	IF pVeData <> 0 THEN
		iDatatypeSize := SIZEOF(ptr^);
		iDatatypeSize := 24;
        ptr := ADR(pVeData^)  +  24  * nVEIndex + (iDatatypeSize * (nArrayIndex));
        ptr^ := val; (* successfully completed return *)
		HLI3_SetVEChannelStringValue := TRUE;
	END_IF
END_IF

END_FUNCTION

// CNC/6 BlockSearch/HLI3_BlockSearch
FUNCTION_BLOCK HLI3_BlockSearch
VAR_INPUT
	/// Number of channel 
	nChanIdx: INT;
	/// interface values 
	BlockSearch: ST_BlockSearch;
END_VAR
VAR_IN_OUT
	/// Edge signal 
	bStartWrite: BOOL;
	/// Edge signal 
	bStartRead: BOOL;
END_VAR
VAR_OUTPUT
	Busy: BOOL;
	Err: BOOL;
	nErrorState: UINT;
	/// interface values 
	nActType: INT;
	fActDistance: LREAL;
	bActAutoReturn: BOOL;
	nActDeviationMax: UDINT;
	nActBlockNumber: DINT;
	nActPass: DINT;
	nActBlockCount: DINT;
	/// current values 
	actualBlockNumber: DINT := 0;
	actualBlockCount: UDINT := 0;
	actualBlockCount_AfterReset: UDINT := 0;
	coveredDistance: DINT;
	coveredDistance_AfterReset: DINT := 0;
END_VAR
VAR
	bReadStarted: BOOL;
	bWriteStarted: BOOL;
	rtStartRead: R_TRIG;
	rtStartWrite: R_TRIG;
	writeType: WriteBsType;
	readType: ReadBsType;
	writeDistance: WriteBsCoveredDistance;
	readDistance: ReadBsCoveredDistance;
	writeAutoReturn: WriteBsAutoReturn;
	readAutoReturn: ReadBsAutoReturn;
	writeDeviationMax: WriteBsDeviationMax;
	readDeviationMax: ReadBsDeviationMax;
	writeBlockNumber: WriteBsBlockNumber;
	ReadBlockNumber: ReadBsBlockNumber;
	writeBlockCount: WriteBsBlockCount;
	ReadBlockCount: ReadBsBlockCount;	
	writePass: WriteBsPass;
	readPass: ReadBsPass;
	nChannelIdxGrp: UDINT;
	/// Timer to read axisposition cyclically        
	Timer: TON;
	actualcoveredDistance: BOOL;
	ChannelMode: UDINT;
	BlockSearchStart: BOOL;
END_VAR

(* ---------------------*----------------------------------|------------------------------------------------------- *)
(* PURPOSE:                                                                                                         *)
(*                                                                                                                  *)
(*                                                                                                                  *)
(* SCOPE:                                                                                                           *)
(*                                                                                                                  *)
(*                                                                                                                  *)
(* REMARKS:                                                                                                         *)
(*                                                                                                                  *)
(*                                                                                                                  *)
(* AUTHOR:              VERSION     DATE                   CHECKED FROM      DATE     STATUS                        *)
(*    MK                1.0         07.05.2003                                                                      *)
(*    TV                1.1         10.06.2006                                                                      *)
(*    TV                1.2         20.08.2014                                                                      *)
(*    TV                1.2         29.09.2014                                                                      *)
(*    TV                1.3         25.06.2015                                                                      *)
(* ---------------------*----------------------------------|------------------------------------------------------- *)

IF NOT HLI3_CheckChannelValid(nChannel := nChanIdx) THEN
	RETURN;
END_IF




Err := FALSE;
nChannelIdxGrp := 16#00020100 + INT_TO_UDINT(nChanIdx)+1;
BlockSearchStart := FALSE;


(* ----------------------------------- *)
(* --- write block search commands --- *)
(* ----------------------------------- *)

rtStartWrite(CLK:=bStartWrite);
IF rtStartWrite.Q THEN
   bWriteStarted := TRUE;
   bStartWrite := FALSE; (* reset the HMI signal *)
END_IF

IF bWriteStarted THEN
   Busy := TRUE;
   IF BlockSearch.nType = 5 THEN
   	BlockSearch.nType := 3;								(* start position by block count *)

		BlockSearch.bAutoReturn := TRUE;
		(*nPass	:= 1;*)
	END_IF

	(* write block search data to memory *)
   writeType(nIdxGrp:=nChannelIdxGrp, bStart:=rtStartWrite.Q, nType:=BlockSearch.nType);
   writeDistance(nIdxGrp:=nChannelIdxGrp, bStart:=rtStartWrite.Q, fDistance:=(BlockSearch.fDistance*10.0));
   writeAutoReturn(nIdxGrp:=nChannelIdxGrp, bStart:=rtStartWrite.Q, bAutoReturn:=BlockSearch.bAutoReturn);
   writeDeviationMax(nIdxGrp:=nChannelIdxGrp, bStart:=rtStartWrite.Q, nDeviationMax:=BlockSearch.nDeviationMax);
   writePass(nIdxGrp:=nChannelIdxGrp, bStart:=rtStartWrite.Q, nPass:=BlockSearch.nPass);

	CASE BlockSearch.nType OF		(* count and number share a part of the memory *)
		3: writeBlockCount(nIdxGrp:=nChannelIdxGrp, bStart:=rtStartWrite.Q, nBlockCount:=BlockSearch.nBlockCount);
		4: writeBlockNumber(nIdxGrp:=nChannelIdxGrp, bStart:=rtStartWrite.Q, nBlockNumber:=BlockSearch.nBlockNumber);
   END_CASE

   IF writeType.Busy = FALSE
      AND writeDistance.BUSY = FALSE
      AND writeAutoReturn.BUSY = FALSE
      AND writeDeviationMax.BUSY = FALSE
      AND writeBlockNumber.BUSY = FALSE
      AND writePass.BUSY = FALSE
      AND writeBlockCount.BUSY = FALSE
   THEN
      Busy := FALSE;
      bWriteStarted := FALSE;
      BlockSearchStart := TRUE;
   END_IF
END_IF


(* Satzsuchlauf starten *)

(*
IF (BlockSearchStart) AND ((nType = 3) OR (nType = 4)) THEN
	PLCMachineMode[nChan].Start := TRUE;
END_IF
*)

(* -------------------------------- *)
(* --- read block search states --- *)
(* -------------------------------- *)

(* the next rows only for test *)
(* Start a cyclic timer with period 2 sec. *)
Timer(IN := NOT(Timer.Q), PT := T#2000ms);

rtStartRead(CLK:=bStartRead);
(*rtStartRead(CLK:=Timer.Q);*)
IF rtStartRead.Q THEN
   bReadStarted := TRUE;
END_IF

IF bReadStarted THEN
	Busy := TRUE;

   readType(nIdxGrp:=nChannelIdxGrp, bStart:=rtStartRead.Q, pDest:=ADR(nActType));
   readDistance(nIdxGrp:=nChannelIdxGrp, bStart:=rtStartRead.Q, pDest:=ADR(fActDistance));
   readAutoReturn(nIdxGrp:=nChannelIdxGrp, bStart:=rtStartRead.Q, pDest:=ADR(bActAutoReturn));
   readDeviationMax(nIdxGrp:=nChannelIdxGrp, bStart:=rtStartRead.Q, pDest:=ADR(nActDeviationMax));
	CASE nActType OF			(* count and number cannot be read within a single cycle! *)
		3: readBlockCount(nIdxGrp:=nChannelIdxGrp, bStart:=rtStartRead.Q, pDest:=ADR(nActBlockCount));
		4: readBlockNumber(nIdxGrp:=nChannelIdxGrp, bStart:=rtStartRead.Q, pDest:=ADR(nActBlockNumber));
	END_CASE;
   readPass(nIdxGrp:=nChannelIdxGrp, bStart:=rtStartRead.Q, pDest:=ADR(nActPass));

   (*
   readActualBlockNumber(nIdxGrp:=nChannelIdxGrp, bStart:=rtStartRead.Q, pDest:=ADR(actualBlockNumber));
   readActualBlockCount(nIdxGrp:=nChannelIdxGrp, bStart:=rtStartRead.Q, pDest:=ADR(actualBlockCount));
   *)

   IF readType.Busy = FALSE
      AND readDistance.Busy = FALSE
      AND readAutoReturn.Busy = FALSE
      AND readDeviationMax.Busy = FALSE
      AND readBlockNumber.Busy = FALSE
      AND readPass.Busy = FALSE      
   THEN
		Busy := FALSE;

		bReadStarted := FALSE;
		bStartRead := FALSE; (* reset the HMI signal *)
   END_IF
END_IF

actualBlockNumber := gpCh[nChanIdx]^.bahn_state.block_nr_r;
actualBlockCount  := gpCh[nChanIdx]^.bahn_state.block_count_r; 

coveredDistance := gpCh[nChanIdx]^.bahn_state.covered_distance_r;  (* just read actual covered distance *)

(* Speichert die Unterbrechungsstelle *)
ChannelMode := HLI3_GetChannelMode(nChanIdx);
IF (actualBlockCount <> 0) AND (ChannelMode = 2) AND (CNCSystem.Channel[nChanIdx].ActState =4) THEN
	actualBlockCount_AfterReset := actualBlockCount;									(* Zeiger bleibt auch nach Reset erhalten *)
	coveredDistance_AfterReset := coveredDistance;
END_IF

(*	UnterbrechungsstelleWeg			:= coveredDistance/10.0;*)

(*actualBlockNumber := gpAx[0]^.lr_state.block_nr_r;  asume first axis is always moved *)


(* handshake during block search on/off *)
gpCh[nChanIdx]^.bahn_lc_control.block_search.enable_w := TRUE;

IF gpCh[nChanIdx]^.bahn_lc_control.block_search.command_r <>
   gpCh[nChanIdx]^.bahn_lc_control.block_search.state_w THEN

   (* acknowledge *)
   gpCh[nChanIdx]^.bahn_lc_control.block_search.state_w :=
      gpCh[nChanIdx]^.bahn_lc_control.block_search.command_r;

(*
   (* pup up of change *)
   IF gpCh[nHliChIfcIdx]^.bahn_lc_control.block_search.state_w THEN
      ADSLOGDINT( msgCtrlMask := ADSLOG_MSGTYPE_MSGBOX OR ADSLOG_MSGTYPE_LOG,
                  msgFmtStr := 'block search: %d', dintArg := 1);
   ELSE
      ADSLOGDINT( msgCtrlMask := ADSLOG_MSGTYPE_MSGBOX OR ADSLOG_MSGTYPE_LOG,
                  msgFmtStr := 'block search: %d', dintArg := 0);
   END_IF
*)
END_IF

END_FUNCTION_BLOCK

// CNC/6 BlockSearch/ReadBlockCount
FUNCTION_BLOCK ReadBlockCount
VAR_INPUT
	nIdxGrp: UDINT;
	bStart: BOOL;
	pDest: POINTER TO DINT;
END_VAR
VAR_OUTPUT
	Busy: BOOL;
	bErr: BOOL;
END_VAR
VAR
	fbRead: ADSREAD;
	bStarted: BOOL;
END_VAR

IF bStarted = FALSE THEN
   IF bStart = TRUE THEN
      bStarted := TRUE;
      bErr := FALSE;
      Busy := TRUE;
   END_IF
END_IF

IF bStarted THEN
   (* raising edge of Timer triggers read request *)
   fbRead( NetID := '', Port := 553, IdxGrp := nIdxGrp, IdxOffs := 16#0000000D,
         LEN := 4, DestAddr := pDest, READ := bStarted, TMOUT := T#1s);
   IF NOT fbRead.Busy THEN
      (* There was an error in the execution of the read request *)
      IF fbRead.Err THEN
         bErr := TRUE;
      END_IF
      fbRead(READ := FALSE);    (* reset because of edge detection in FB ADSREAD *)
      bStarted := FALSE;
      Busy := FALSE;
   END_IF
END_IF

END_FUNCTION_BLOCK

// CNC/6 BlockSearch/ReadBlockNumber
FUNCTION_BLOCK ReadBlockNumber
VAR_INPUT
	nIdxGrp: UDINT;
	bStart: BOOL;
	pDest: POINTER TO DINT;
END_VAR
VAR_OUTPUT
	Busy: BOOL;
	bErr: BOOL;
END_VAR
VAR
	fbRead: ADSREAD;
	bStarted: BOOL;
END_VAR

IF bStarted = FALSE THEN
   IF bStart = TRUE THEN
      bStarted := TRUE;
      bErr := FALSE;
      Busy := TRUE;
   END_IF
END_IF

IF bStarted THEN
   (* raising edge of Timer triggers read request *)
   fbRead( NetID := '', Port := 553, IdxGrp := nIdxGrp, IdxOffs := 16#0000000E,
         LEN := 4, DestAddr := pDest, READ := bStarted, TMOUT := T#1s);
   IF NOT fbRead.Busy THEN
      (* There was an error in the execution of the read request *)
      IF fbRead.Err THEN
         bErr := TRUE;
      END_IF
      fbRead(READ := FALSE);    (* reset because of edge detection in FB ADSREAD *)
      bStarted := FALSE;
      Busy := FALSE;
   END_IF
END_IF

END_FUNCTION_BLOCK

// CNC/6 BlockSearch/WriteBsType
FUNCTION_BLOCK WriteBsType
VAR_INPUT
	nIdxGrp: UDINT;
	bStart: BOOL;
	nType: UINT;
END_VAR
VAR_OUTPUT
	Busy: BOOL;
	bErr: BOOL;
END_VAR
VAR
	fbWrite: ADSWRITE;
	bStarted: BOOL;
END_VAR

IF bStarted = FALSE THEN
   IF bStart = TRUE THEN
      bStarted := TRUE;
      bErr := FALSE;
      Busy := TRUE;
   END_IF
END_IF

IF bStarted THEN
   (* raising edge of Timer triggers write request *)
   fbWrite( NetID := '', Port := 553, IdxGrp := nIdxGrp, IdxOffs := 16#00000049,
         LEN := 2, SrcAddr := ADR(nType), WRITE := bStarted, TMOUT := T#1s);
   IF NOT fbWrite.Busy THEN
      (* There was an error in the execution of the write request *)
      IF fbWrite.Err THEN
         bErr := TRUE;
      END_IF
      fbWrite(WRITE := FALSE);    (* reset because of edge detection in FB ADSWRITE *)
      bStarted := FALSE;
      Busy := FALSE;
   END_IF
END_IF

END_FUNCTION_BLOCK

// CNC/6 BlockSearch/ReadBsType
FUNCTION_BLOCK ReadBsType
VAR_INPUT
	nIdxGrp: UDINT;
	bStart: BOOL;
	pDest: POINTER TO UINT;
END_VAR
VAR_OUTPUT
	Busy: BOOL;
	bErr: BOOL;
END_VAR
VAR
	fbRead: ADSREAD;
	bStarted: BOOL;
END_VAR

IF bStarted = FALSE THEN
   IF bStart = TRUE THEN
      bStarted := TRUE;
      bErr := FALSE;
      Busy := TRUE;
   END_IF
END_IF

IF bStarted THEN
   (* raising edge of Timer triggers read request *)
   fbRead( NetID := '', Port := 553, IdxGrp := nIdxGrp, IdxOffs := 16#00000061,
         LEN := 2, DestAddr := pDest, READ := bStarted, TMOUT := T#1s);
   IF NOT fbRead.Busy THEN
      (* There was an error in the execution of the read request *)
      IF fbRead.Err THEN
         bErr := TRUE;
      END_IF
      fbRead(READ := FALSE);    (* reset because of edge detection in FB ADSREAD *)
      bStarted := FALSE;
      Busy := FALSE;
   END_IF
END_IF

END_FUNCTION_BLOCK

// CNC/6 BlockSearch/WriteBsCoveredDistance
FUNCTION_BLOCK WriteBsCoveredDistance
VAR_INPUT
	nIdxGrp: UDINT;
	bStart: BOOL;
	fDistance: LREAL;
END_VAR
VAR_OUTPUT
	Busy: BOOL;
	bErr: BOOL;
END_VAR
VAR
	fbWrite: ADSWRITE;
	bStarted: BOOL;
END_VAR

IF bStarted = FALSE THEN
   IF bStart = TRUE THEN
      bStarted := TRUE;
      bErr := FALSE;
      Busy := TRUE;
   END_IF
END_IF

IF bStarted THEN
   (* raising edge of Timer triggers write request *)
   fbWrite( NetID := '', Port := 553, IdxGrp := nIdxGrp, IdxOffs := 16#0000004A,
         LEN := 8, SrcAddr := ADR(fDistance), WRITE := bStarted, TMOUT := T#1s);
   IF NOT fbWrite.Busy THEN
      (* There was an error in the execution of the write request *)
      IF fbWrite.Err THEN
         bErr := TRUE;
      END_IF
      fbWrite(WRITE := FALSE);    (* reset because of edge detection in FB ADSWRITE *)
      bStarted := FALSE;
      Busy := FALSE;
   END_IF
END_IF

END_FUNCTION_BLOCK

// CNC/6 BlockSearch/ReadBsCoveredDistance
FUNCTION_BLOCK ReadBsCoveredDistance
VAR_INPUT
	nIdxGrp: UDINT;
	bStart: BOOL;
	pDest: POINTER TO LREAL;
END_VAR
VAR_OUTPUT
	Busy: BOOL;
	bErr: BOOL;
END_VAR
VAR
	fbRead: ADSREAD;
	bStarted: BOOL;
END_VAR

IF bStarted = FALSE THEN
   IF bStart = TRUE THEN
      bStarted := TRUE;
      bErr := FALSE;
      Busy := TRUE;
   END_IF
END_IF

IF bStarted THEN
   (* raising edge of Timer triggers read request *)
   fbRead( NetID := '', Port := 553, IdxGrp := nIdxGrp, IdxOffs := 16#00000062,
         LEN := 8, DestAddr := pDest, READ := bStarted, TMOUT := T#1s);
   IF NOT fbRead.Busy THEN
      (* There was an error in the execution of the read request *)
      IF fbRead.Err THEN
         bErr := TRUE;
      END_IF
      fbRead(READ := FALSE);    (* reset because of edge detection in FB ADSREAD *)
      bStarted := FALSE;
      Busy := FALSE;
   END_IF
END_IF

END_FUNCTION_BLOCK

// CNC/6 BlockSearch/WriteBsAutoReturn
FUNCTION_BLOCK WriteBsAutoReturn
VAR_INPUT
	nIdxGrp: UDINT;
	bStart: BOOL;
	bAutoReturn: BOOL;
END_VAR
VAR_OUTPUT
	Busy: BOOL;
	bErr: BOOL;
END_VAR
VAR
	fbWrite: ADSWRITE;
	bStarted: BOOL;
END_VAR

IF bStarted = FALSE THEN
   IF bStart = TRUE THEN
      bStarted := TRUE;
      bErr := FALSE;
      Busy := TRUE;
   END_IF
END_IF

IF bStarted THEN
   (* raising edge of Timer triggers write request *)
   fbWrite( NetID := '', Port := 553, IdxGrp := nIdxGrp, IdxOffs := 16#0000004B,
         LEN := 1, SrcAddr := ADR(bAutoReturn), WRITE := bStarted, TMOUT := T#1s);
   IF NOT fbWrite.Busy THEN
      (* There was an error in the execution of the write request *)
      IF fbWrite.Err THEN
         bErr := TRUE;
      END_IF
      fbWrite(WRITE := FALSE);    (* reset because of edge detection in FB ADSWRITE *)
      bStarted := FALSE;
      Busy := FALSE;
   END_IF
END_IF

END_FUNCTION_BLOCK

// CNC/6 BlockSearch/ReadBsAutoReturn
FUNCTION_BLOCK ReadBsAutoReturn
VAR_INPUT
	nIdxGrp: UDINT;
	bStart: BOOL;
	pDest: POINTER TO BOOL;
END_VAR
VAR_OUTPUT
	Busy: BOOL;
	bErr: BOOL;
END_VAR
VAR
	fbRead: ADSREAD;
	bStarted: BOOL;
END_VAR

IF bStarted = FALSE THEN
   IF bStart = TRUE THEN
      bStarted := TRUE;
      bErr := FALSE;
      Busy := TRUE;
   END_IF
END_IF

IF bStarted THEN
   (* raising edge of Timer triggers read request *)
   fbRead( NetID := '', Port := 553, IdxGrp := nIdxGrp, IdxOffs := 16#00000063,
         LEN := 1, DestAddr := pDest, READ := bStarted, TMOUT := T#1s);
   IF NOT fbRead.Busy THEN
      (* There was an error in the execution of the read request *)
      IF fbRead.Err THEN
         bErr := TRUE;
      END_IF
      fbRead(READ := FALSE);    (* reset because of edge detection in FB ADSREAD *)
      bStarted := FALSE;
      Busy := FALSE;
   END_IF
END_IF

END_FUNCTION_BLOCK

// CNC/6 BlockSearch/WriteBsDeviationMax
FUNCTION_BLOCK WriteBsDeviationMax
VAR_INPUT
	nIdxGrp: UDINT;
	bStart: BOOL;
	nDeviationMax: UDINT;
END_VAR
VAR_OUTPUT
	Busy: BOOL;
	bErr: BOOL;
END_VAR
VAR
	fbWrite: ADSWRITE;
	bStarted: BOOL;
END_VAR

IF bStarted = FALSE THEN
   IF bStart = TRUE THEN
      bStarted := TRUE;
      bErr := FALSE;
      Busy := TRUE;
   END_IF
END_IF

IF bStarted THEN
   (* raising edge of Timer triggers write request *)
   fbWrite( NetID := '', Port := 553, IdxGrp := nIdxGrp, IdxOffs := 16#0000004C,
         LEN := 4, SrcAddr := ADR(nDeviationMax), WRITE := bStarted, TMOUT := T#1s);
   IF NOT fbWrite.Busy THEN
      (* There was an error in the execution of the write request *)
      IF fbWrite.Err THEN
         bErr := TRUE;
      END_IF
      fbWrite(WRITE := FALSE);    (* reset because of edge detection in FB ADSWRITE *)
      bStarted := FALSE;
      Busy := FALSE;
   END_IF
END_IF

END_FUNCTION_BLOCK

// CNC/6 BlockSearch/ReadBsDeviationMax
FUNCTION_BLOCK ReadBsDeviationMax
VAR_INPUT
	nIdxGrp: UDINT;
	bStart: BOOL;
	pDest: POINTER TO UDINT;
END_VAR
VAR_OUTPUT
	Busy: BOOL;
	bErr: BOOL;
END_VAR
VAR
	fbRead: ADSREAD;
	bStarted: BOOL;
END_VAR

IF bStarted = FALSE THEN
   IF bStart = TRUE THEN
      bStarted := TRUE;
      bErr := FALSE;
      Busy := TRUE;
   END_IF
END_IF

IF bStarted THEN
   (* raising edge of Timer triggers read request *)
   fbRead( NetID := '', Port := 553, IdxGrp := nIdxGrp, IdxOffs := 16#00000064,
         LEN := 4, DestAddr := pDest, READ := bStarted, TMOUT := T#1s);
   IF NOT fbRead.Busy THEN
      (* There was an error in the execution of the read request *)
      IF fbRead.Err THEN
         bErr := TRUE;
      END_IF
      fbRead(READ := FALSE);    (* reset because of edge detection in FB ADSREAD *)
      bStarted := FALSE;
      Busy := FALSE;
   END_IF
END_IF

END_FUNCTION_BLOCK

// CNC/6 BlockSearch/WriteBsBlockNumber
FUNCTION_BLOCK WriteBsBlockNumber
VAR_INPUT
	nIdxGrp: UDINT;
	bStart: BOOL;
	nBlockNumber: DINT;
END_VAR
VAR_OUTPUT
	Busy: BOOL;
	bErr: BOOL;
END_VAR
VAR
	fbWrite: ADSWRITE;
	bStarted: BOOL;
END_VAR

IF bStarted = FALSE THEN
   IF bStart = TRUE THEN
      bStarted := TRUE;
      bErr := FALSE;
      Busy := TRUE;
   END_IF
END_IF

IF bStarted THEN
   (* raising edge of Timer triggers write request *)
   fbWrite( NetID := '', Port := 553, IdxGrp := nIdxGrp, IdxOffs := 16#0000005F,
         LEN := 4, SrcAddr := ADR(nBlockNumber), WRITE := bStarted, TMOUT := T#1s);
   IF NOT fbWrite.Busy THEN
      (* There was an error in the execution of the write request *)
      IF fbWrite.Err THEN
         bErr := TRUE;
      END_IF
      fbWrite(WRITE := FALSE);    (* reset because of edge detection in FB ADSWRITE *)
      bStarted := FALSE;
      Busy := FALSE;
   END_IF
END_IF

END_FUNCTION_BLOCK

// CNC/6 BlockSearch/ReadBsBlockNumber
FUNCTION_BLOCK ReadBsBlockNumber
VAR_INPUT
	nIdxGrp: UDINT;
	bStart: BOOL;
	pDest: POINTER TO DINT;
END_VAR
VAR_OUTPUT
	Busy: BOOL;
	bErr: BOOL;
END_VAR
VAR
	fbRead: ADSREAD;
	bStarted: BOOL;
END_VAR

IF bStarted = FALSE THEN
   IF bStart = TRUE THEN
      bStarted := TRUE;
      bErr := FALSE;
      Busy := TRUE;
   END_IF
END_IF

IF bStarted THEN
   (* raising edge of Timer triggers read request *)
   fbRead( NetID := '', Port := 553, IdxGrp := nIdxGrp, IdxOffs := 16#00000077,
         LEN := 4, DestAddr := pDest, READ := bStarted, TMOUT := T#1s);
   IF NOT fbRead.Busy THEN
      (* There was an error in the execution of the read request *)
      IF fbRead.Err THEN
         bErr := TRUE;
      END_IF
      fbRead(READ := FALSE);    (* reset because of edge detection in FB ADSREAD *)
      bStarted := FALSE;
      Busy := FALSE;
   END_IF
END_IF

END_FUNCTION_BLOCK

// CNC/6 BlockSearch/WriteBsBlockCount
FUNCTION_BLOCK WriteBsBlockCount
VAR_INPUT
	nIdxGrp: UDINT;
	bStart: BOOL;
	nBlockCount: DINT;
END_VAR
VAR_OUTPUT
	Busy: BOOL;
	bErr: BOOL;
END_VAR
VAR
	fbWrite: ADSWRITE;
	bStarted: BOOL;
END_VAR

IF bStarted = FALSE THEN
   IF bStart = TRUE THEN
      bStarted := TRUE;
      bErr := FALSE;
      Busy := TRUE;
   END_IF
END_IF

IF bStarted THEN
   (* raising edge of Timer triggers write request *)
   fbWrite( NetID := '', Port := 553, IdxGrp := nIdxGrp, IdxOffs := 16#0000005E,
         LEN := 4, SrcAddr := ADR(nBlockCount), WRITE := bStarted, TMOUT := T#1s);
   IF NOT fbWrite.Busy THEN
      (* There was an error in the execution of the write request *)
      IF fbWrite.Err THEN
         bErr := TRUE;
      END_IF
      fbWrite(WRITE := FALSE);    (* reset because of edge detection in FB ADSWRITE *)
      bStarted := FALSE;
      Busy := FALSE;
   END_IF
END_IF

END_FUNCTION_BLOCK

// CNC/6 BlockSearch/ReadBsBlockCount
FUNCTION_BLOCK ReadBsBlockCount
VAR_INPUT
	nIdxGrp: UDINT;
	bStart: BOOL;
	pDest: POINTER TO DINT;
END_VAR
VAR_OUTPUT
	Busy: BOOL;
	bErr: BOOL;
END_VAR
VAR
	fbRead: ADSREAD;
	bStarted: BOOL;
END_VAR

IF bStarted = FALSE THEN
   IF bStart = TRUE THEN
      bStarted := TRUE;
      bErr := FALSE;
      Busy := TRUE;
   END_IF
END_IF

IF bStarted THEN
   (* raising edge of Timer triggers read request *)
   fbRead( NetID := '', Port := 553, IdxGrp := nIdxGrp, IdxOffs := 16#00000076,
         LEN := 4, DestAddr := pDest, READ := bStarted, TMOUT := T#1s);
   IF NOT fbRead.Busy THEN
      (* There was an error in the execution of the read request *)
      IF fbRead.Err THEN
         bErr := TRUE;
      END_IF
      fbRead(READ := FALSE);    (* reset because of edge detection in FB ADSREAD *)
      bStarted := FALSE;
      Busy := FALSE;
   END_IF
END_IF

END_FUNCTION_BLOCK

// CNC/6 BlockSearch/WriteBsPass
FUNCTION_BLOCK WriteBsPass
VAR_INPUT
	nIdxGrp: UDINT;
	bStart: BOOL;
	nPass: DINT;
END_VAR
VAR_OUTPUT
	Busy: BOOL;
	bErr: BOOL;
END_VAR
VAR
	fbWrite: ADSWRITE;
	bStarted: BOOL;
END_VAR

IF bStarted = FALSE THEN
   IF bStart = TRUE THEN
      bStarted := TRUE;
      bErr := FALSE;
      Busy := TRUE;
   END_IF
END_IF

IF bStarted THEN
   (* raising edge of Timer triggers write request *)
   fbWrite( NetID := '', Port := 553, IdxGrp := nIdxGrp, IdxOffs := 16#00000060,
         LEN := 4, SrcAddr := ADR(nPass), WRITE := bStarted, TMOUT := T#1s);
   IF NOT fbWrite.Busy THEN
      (* There was an error in the execution of the write request *)
      IF fbWrite.Err THEN
         bErr := TRUE;
      END_IF
      fbWrite(WRITE := FALSE);    (* reset because of edge detection in FB ADSWRITE *)
      bStarted := FALSE;
      Busy := FALSE;
   END_IF
END_IF

END_FUNCTION_BLOCK

// CNC/6 BlockSearch/ReadBsPass
FUNCTION_BLOCK ReadBsPass
VAR_INPUT
	nIdxGrp: UDINT;
	bStart: BOOL;
	pDest: POINTER TO DINT;
END_VAR
VAR_OUTPUT
	Busy: BOOL;
	bErr: BOOL;
END_VAR
VAR
	fbRead: ADSREAD;
	bStarted: BOOL;
END_VAR

IF bStarted = FALSE THEN
   IF bStart = TRUE THEN
      bStarted := TRUE;
      bErr := FALSE;
      Busy := TRUE;
   END_IF
END_IF

IF bStarted THEN
   (* raising edge of Timer triggers read request *)
   fbRead( NetID := '', Port := 553, IdxGrp := nIdxGrp, IdxOffs := 16#00000078,
         LEN := 4, DestAddr := pDest, READ := bStarted, TMOUT := T#1s);
   IF NOT fbRead.Busy THEN
      (* There was an error in the execution of the read request *)
      IF fbRead.Err THEN
         bErr := TRUE;
      END_IF
      fbRead(READ := FALSE);    (* reset because of edge detection in FB ADSREAD *)
      bStarted := FALSE;
      Busy := FALSE;
   END_IF
END_IF

END_FUNCTION_BLOCK

// CNC/8 Mis/FB_WriteCNCZeroOffset
/// ------------------------------------------------------------------------------------ 
/// Desc:	Description																	
///**************************************************************************************
///**************************************************************************************
///	 Write NPV Value directly to CNC core using V.G. Variables via ADS	
///**************************************************************************************
FUNCTION_BLOCK FB_WriteCNCZeroOffset
VAR_INPUT
	/// rising edge to start 
	bExecute: BOOL;
	/// which table, G54=1, G55=2, G55=3, .... 
	nG159Index: BYTE;
	/// Channel Indedx
	nChanIdx: UDINT;
	/// Axis name in channel 
	sAxisName: STRING(95);
	/// value to set 
	lrValue: LREAL;
END_VAR
VAR_OUTPUT
	bBusy: BOOL;
	bError: BOOL;
	nErrorID: UDINT;
END_VAR
VAR
	fbAdsWrite: ADSWRITE;
	stCNCG159VG: ST_CNCG159VG;
END_VAR

stCNCG159VG.dValue := LREAL_TO_DINT(lrValue * 10000);
stCNCG159VG.sTarget := 'V.G.NP[';
stCNCG159VG.sTarget := CONCAT(stCNCG159VG.sTarget, BYTE_TO_STRING(nG159Index));
stCNCG159VG.sTarget := CONCAT(stCNCG159VG.sTarget, '].V.');
stCNCG159VG.sTarget := CONCAT(stCNCG159VG.sTarget,sAxisName);

fbAdsWrite(
	PORT:= 552 ,
	IDXGRP:= 16#22300 + nChanIdx+1,
	IDXOFFS:=16#3F,
	LEN:= SIZEOF(stCNCG159VG) ,
	SRCADDR:=ADR(stCNCG159VG) ,
	WRITE:= bExecute,
	TMOUT:= ,
	BUSY=> bBusy,
	ERR=> bError ,
	ERRID=> nErrorID);

END_FUNCTION_BLOCK

// CNC/8 Mis/FB_WriteCNCZeroOffsetDefault
/// ------------------------------------------------------------------------------------ 
/// Desc:	Description																	
///**************************************************************************************
///**************************************************************************************
///	 Write NPV Default (the active table afetr reset) directly to CNC core using V.G. Variables via ADS	
///**************************************************************************************
FUNCTION_BLOCK FB_WriteCNCZeroOffsetDefault
VAR_INPUT
	/// rising edge to start 
	bExecute: BOOL;
	/// which table, G54=1, G55=2, G55=3, .... 
	nG159Index: BYTE;
	/// Channel Indedx
	nChanIdx: UDINT;
END_VAR
VAR_OUTPUT
	bBusy: BOOL;
	bError: BOOL;
	nErrorID: UDINT;
END_VAR
VAR
	fbAdsWrite: ADSWRITE;
	stCNCG159VG: ST_CNCG159VG;
END_VAR

stCNCG159VG.dValue := nG159Index;
stCNCG159VG.sTarget := 'V.G.NP_DEFAULT';

fbAdsWrite(
	PORT:= 552 ,
	IDXGRP:= 16#22300 + nChanIdx+1,
	IDXOFFS:=16#3F,
	LEN:= SIZEOF(stCNCG159VG) ,
	SRCADDR:=ADR(stCNCG159VG) ,
	WRITE:= bExecute,
	TMOUT:= ,
	BUSY=> bBusy,
	ERR=> bError ,
	ERRID=> nErrorID);

END_FUNCTION_BLOCK

// CNC/8 Mis/HLI_HandleMessages
FUNCTION_BLOCK HLI_HandleMessages
VAR_INPUT
	/// Enable 
	bEnable: BOOL;
	/// Number of channel 
	nChanIdx: INT;
	/// Channelstruct 
	pChannel: POINTER TO ST_CncChannel;
END_VAR
VAR_OUTPUT
	bNewMessage: BOOL;
	bError: BOOL;
	sMessage: STRING(255);
END_VAR
VAR
	/// Index of channel specific HLI area 

	bFirstCycle: BOOL := TRUE;
	bModeChanged: BOOL;
	nState: USINT;
	nActMode: UDINT;
	dwCncState: DWORD;
	fbRtrigStateStart: R_TRIG;
	pString: POINTER TO STRING(HLI_MSG_CONTENT_STRL);
	fbLog: ADSLOGEVENT;
	stMessageData: TcEvent;
END_VAR
VAR CONSTANT
	sFormat: STRING(2) := '%s';
END_VAR

(******************************************************************************)
(* Name:		HLI_HandleMessages											 	*)
(* Date:		08/12/01													 	*)
(* Author:	H. Rausch (Beckhoff Automation GmbH)							 	*)
(* Ver:		1.0																	*)
(* Desc:		Function block for recieving messages from CNC and passing them to*)
(*				the TwinCAT EventLogger. Only the latest message from CNC is 	*)
(*				active there. The event will be resetted if a new message from	*)
(*				CNC is recieved, the CNC state changes to 'ACTIVE', the CNC mode*)
(*				is changed or the channel is resetted							*)
(*																				*)
(*				Messages are passed as a fill string to the event logger with 	*)
(*				source id 9000 and event id 1. This requires a correspondant 	*)
(*				configuration in the tceventsourcelocation.xml and in an		*)
(*				associated message file!										*)
(* ---------------------------------------------------------------------------*)
(* Rev:		Add new version number here!										*)
(* Date.		Add revision data here											*)
(* Desc:		Add revision description here!									*)
(******************************************************************************)

(* Write event config data once on start up *)
IF bFirstCycle THEN
	stMessageData.bQuitRequired			:= TRUE;
	stMessageData.Class					:= TCEVENTCLASS_MESSAGE;
	stMessageData.DataFormatStrAddress	:= ADR(sFormat);
	stMessageData.Prio					:= 0;
	stMessageData.Id					:= 1;
	stMessageData.SourceId 				:= 9000;
	stMessageData.Flags 				:= TCEVENTFLAG_LOG OR TCEVENTFLAG_SRCID;
	stMessageData.StreamType			:= TCEVENTSTREAM_SIMPLE;
	stMessageData.ProgId 				:= 'TcEventFormatter.TcXmlFormatter';
END_IF



(* Check for zero pointer and leave fb if necessary *)
IF NOT HLI3_CheckChannelValid(nChannel := nChanIdx) THEN
	RETURN;
END_IF
	(* Check CNC state *)
	dwCncState := HLI3_GetChannelState(nChanIdx:=nChanIdx);

	(* Rising trig if CNC state changes to ACTIVE *)
	fbRtrigStateStart
		(CLK := (dwCncState = HLI_IMCM_PROCESS_ACTIVE));

	(* Watch CNC mode *)
	bModeChanged	:= (nActMode <> pChannel^.ActMode);
	nActMode 		:= pChannel^.ActMode;

IF NOT bEnable THEN
	gpCh[nChanIdx]^.msg_mc_control.enable_w				:= FALSE;
	gpCh[nChanIdx]^.msg_mc_control.request_semaphor_rw	:= FALSE;
	sMessage										:= '';
ELSE
	gpCh[nChanIdx]^.msg_mc_control.enable_w 			:= TRUE;

	CASE nState OF
	 0:
		(* Wait for new messages from CNC *)
		IF gpCh[nChanIdx]^.msg_mc_control.request_semaphor_rw THEN
			(* Convert byte stream to string *)
			pString  := ADR(gpCh[nChanIdx]^.msg_mc_control.request_r.inhalt);
			sMessage := pString^;
			(* Reset notification from HLI *)
			gpCh[nChanIdx]^.msg_mc_control.request_semaphor_rw := FALSE;

			nState := 1;
		END_IF

	 1:
		(* Wait that ADSEVENTLOG instance is cleared *)
		IF (fbLog.EventState = 0) THEN
			nState := 2;
		END_IF

	 2:
		(* Set message to eventlogger *)
		IF (fbLog.EventState > 0) THEN
			nState := 0;
		END_IF

	END_CASE

	(* Managing Eventlogger *)
	fbLog
		(NETID				:= '',
		 PORT					:= 110,
		 Event				:= (nState = 2),
		 EventQuit			:= (nState = 1) OR
									(dwCncState = HLI_IMCM_PROCESS_RESETTING) OR
									fbRtrigStateStart.Q OR
									bModeChanged,
		 EventConfigData	:= stMessageData,
		 EventDataAddress	:= ADR(sMessage),
		 EventDataLength	:= SIZEOF(sMessage),
		 TMOUT				:= t#2s
		);
END_IF

(* Reset first cycle indicator *)
bFirstCycle := FALSE;

END_FUNCTION_BLOCK

// CNC/8 Mis/HLI3_CheckCNCAlive
PROGRAM HLI3_CheckCNCAlive
VAR_INPUT
	nChanIdx: INT;
END_VAR

VAR
	bMessageDisplayed : BOOL;
END_VAR

(* The assumption is made that the cycle time of the PLC is at least twice as big as the CNC cycle time.

The Cycle time of CNC is displayed in element:
	pMC[1]^.addr^.HLIHeadChannel_Data.LCWatchDogUnit_lc.D_cycle_time_r

remark: Take care if PLC cycle is smaller not to check CNC faster as possible !!!

To simulate failure of CNC set cycle time of PLC smaller than CNC (Resource/task configuration).
*)

// HLI3_CheckCNCAlive := FALSE;
IF NOT HLI3_CheckChannelValid(nChannel := nChanIdx) THEN
	RETURN;
END_IF
 
(* Copy current state of live sign to watchdog state    *)
gpCh[nChanIdx]^.head.lc_watchdog.alive_rw
	:= gpCh[nChanIdx]^.head.lc_watchdog.alive_rw;

IF gpCh[nChanIdx]^.head.lc_watchdog.alive_rw = FALSE AND NOT bMessageDisplayed THEN
	(* PLC detects CNC not alive -> start individual emergency stop within PLC *)
	ADSLOGSTR( msgCtrlMask := ADSLOG_MSGTYPE_ERROR OR
							ADSLOG_MSGTYPE_MSGBOX OR
							ADSLOG_MSGTYPE_LOG,
			msgFmtStr := 'PLC detects CNC not alive: %s',
			strArg := 'channel 1');
			
			bMessageDisplayed := TRUE;
END_IF


(* assign return value *)
//HLI3_CheckCNCAlive := gpCh[nChanIdx]^.head.lc_watchdog.alive_rw;

(* reset live sign for next cycle *)
gpCh[nChanIdx]^.head.lc_watchdog.alive_rw := FALSE;

END_PROGRAM

// CNC/8 Mis/HLI3_GetLogAxisId
FUNCTION HLI3_GetLogAxisId : INT
VAR_INPUT
	nHliAxisIdx: INT;
END_VAR
VAR
	i: INT;
END_VAR

(* ========================================================= *)
(*    FUN: HLI3_GetLogAxisId                            	 *)
(* --------------------------------------------------------- *)
(*   Desc: returns the Log. Axis Idx for a given HLI Index   *)
(*   Author: TV                                              *)
(*   Date: 22.01.2014                                        *)
(*   Rev.: 1.0                                               *)
(* ========================================================= *)
HLI3_GetLogAxisId := -1;
IF NOT HLI3_CheckAxisValid(nHliAxisIdx := nHliAxisIdx) THEN
	RETURN;
END_IF

HLI3_GetLogAxisId := UINT_TO_INT(gpAx[nHliAxisIdx]^.head.log_ax_nr_r);

END_FUNCTION

// DUTs/CNC_DataTyps/ITF_ToolAction
INTERFACE ITF_ToolAction

/// Commits the tool data transfer action if it returns true
METHOD Commit : BOOL
VAR_INPUT
	t : ST_CNC_TOOL_DATA_EXT;
END_VAR
END_METHOD

PROPERTY Tool : ST_CNC_TOOL_DATA_EXT
GET
END_GET
END_PROPERTY

END_INTERFACE

// DUTs/ManualFnc/FB_ManualFncBody
{attribute 'OPC.UA.DA' := '1'}
FUNCTION_BLOCK FB_ManualFncBody EXTENDS FB_ManualFncLite
VAR_INPUT
	headerText				:  	STRING;
	addText					:  	STRING;
	sort					:	UDINT;
	hide					:	ST_FncHide;
	cssAttribut				:	STRING;
	infoText1				:	STRING;
	infoText2				:	STRING;
	infoText3				:	STRING;
	infoText4				:	STRING;
	error					:	BOOL;
	select					:	BOOL;
END_VAR

END_FUNCTION_BLOCK

// DUTs/ManualFnc/FB_ManualFncLite
{attribute 'OPC.UA.DA' := '1'}
FUNCTION_BLOCK FB_ManualFncLite
VAR CONSTANT
	{attribute 'const_non_replaced'}
	hmiElementId			:	STRING := 'HMI_FNC';
END_VAR

//			Left				Visibility 5x / Error/select				right
//	 ___________________________________________________________________________________
//	|				| l |                                            |r |				|
//	|               | e |      headerText :  addText                 |i |               |
//	|  	 /          | f |--------------------------------------------|g |          \   	|
//	|	/           | t |    infoText1   		|	infoText2		 |ht|           \  	|		
//  |	\           | . |                       |                    |. |           /   |
//  | 	 \          | st|--------------------------------------------|st|          /    |
// 	| Left.key.text	| at|    infoText3          |	infoText4        |at| right.key.text|
//	|_______________|_us|_______________________|____________________|us|_______________|

// sort  [1 - n] änder die Anzeige Reihenfolge

END_FUNCTION_BLOCK

// DUTs/ManualFnc/FB_ManualFncFull
{attribute 'OPC.UA.DA' := '1'}
FUNCTION_BLOCK FB_ManualFncFull EXTENDS FB_ManualFncBody
VAR_INPUT
	left					:	FB_ManualFncKey;
	right					:	FB_ManualFncKey;
END_VAR

//			Left				Visibility 5x / Error/select				right
//	 ___________________________________________________________________________________
//	|				| l |                                            |r |				|
//	|               | e |      headerText :  addText                 |i |               |
//	|  	 /          | f |--------------------------------------------|g |          \   	|
//	|	/           | t |    infoText1   		|	infoText2		 |ht|           \  	|		
//  |	\           | . |                       |                    |. |           /   |
//  | 	 \          | st|--------------------------------------------|st|          /    |
// 	| Left.key.text	| at|    infoText3          |	infoText4        |at| right.key.text|
//	|_______________|_us|_______________________|____________________|us|_______________|

// sort  [1 - n] änder die Anzeige Reihenfolge

END_FUNCTION_BLOCK

// DUTs/ManualFnc/FB_ManualFncKey
{attribute 'OPC.UA.DA' := '1'}
FUNCTION_BLOCK FB_ManualFncKey
VAR_INPUT
	key					:	FB_ManualFncKeyBasic;
	status				:	FB_ManualFncStatus;
END_VAR

END_FUNCTION_BLOCK

// DUTs/ManualFnc/FB_ManualFncKeyBasic
{attribute 'OPC.UA.DA' := '1'}
FUNCTION_BLOCK FB_ManualFncKeyBasic
VAR_INPUT
	text				:	STRING;
	disable				:	BOOL;
	userLevel			:	INT;
	liveBit				:	BOOL;
	q					:	BOOL;
	colorChange			:	BOOL := FALSE;
	hide				:	ST_KeyHide;	
END_VAR

END_FUNCTION_BLOCK

// DUTs/ManualFnc/FB_ManualFncStatus
{attribute 'OPC.UA.DA' := '1'}
FUNCTION_BLOCK FB_ManualFncStatus
VAR_INPUT
	text				:	STRING;
	colorChange			:	BOOL := FALSE;
	hide				:	ST_StatusHide;	
END_VAR

END_FUNCTION_BLOCK
